FUNCTION Convert_DT_TO_LWORD : Hresult
VAR_INPUT
	in : DT;
	out : REFERENCE TO LWORD;
END_VAR
VAR
	converted : LWORD;
END_VAR

converted := DT_TO_LWORD(in);

IF (LWORD_TO_DT(converted) <> in) THEN
	Convert_DT_TO_LWORD := INCOMPATIBLE;
	RETURN;
END_IF

out := converted;

END_FUNCTION

(* stored: Version 1.1.0.1, ProductVersion 3.1.4024.12
   POU Convert_DT_TO_LWORD: Id {5503b576-0c6b-4ca7-9624-b86651e416dc}, SpecialFunc None *)
